FUNCTION n08b2BYTE
  (* Standard: 61499-1 *)
  (* Version 1.0, 2024-02-22, franz *)
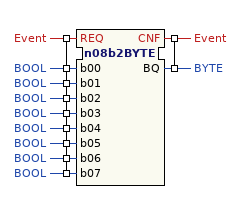
  EVENT_INPUT
    REQ WITH b00, b01, b02, b03, b04, b05, b06, b07;
  END_EVENT
  EVENT_OUTPUT
    CNF WITH BQ;
  END_EVENT
  VAR_INPUT
    b00 : BOOL; (* BIT 00 *)
    b01 : BOOL; (* BIT 01 *)
    b02 : BOOL; (* BIT 02 *)
    b03 : BOOL; (* BIT 03 *)
    b04 : BOOL; (* BIT 04 *)
    b05 : BOOL; (* BIT 05 *)
    b06 : BOOL; (* BIT 06 *)
    b07 : BOOL; (* BIT 07 *)
  END_VAR
  VAR_OUTPUT
    BQ : BYTE;
  END_VAR
  BODY IN ST:
FUNCTION n08b2BYTE

VAR_INPUT
	b00 : BOOL;    // BIT 00
	b01 : BOOL;    // BIT 01
	b02 : BOOL;    // BIT 02
	b03 : BOOL;    // BIT 03
	b04 : BOOL;    // BIT 04
	b05 : BOOL;    // BIT 05
	b06 : BOOL;    // BIT 06
	b07 : BOOL;    // BIT 07
END_VAR

VAR_OUTPUT
	BQ : BYTE;
END_VAR

END_FUNCTION
  END_BODY
END_FUNCTION
